FUNCTION F_Counter : BOOL

VAR_INPUT
	eCounterMode : E_CounterMode;
END_VAR
VAR_IN_OUT
	stCounter	: ST_Counter_Item;//ST_Conunter;
END_VAR
VAR
END_VAR

IF (eCounterMode = E_CounterMode.eCounterMode_Ok_Up) THEN
	stCounter.nValueOk:=stCounter.nValueOk+1;
	stCounter.nValueSerialError:=0;
ELSIF (eCounterMode = E_CounterMode.eCounterMode_Ok_Down) THEN	
	stCounter.nValueOk:=stCounter.nValueOk-1;
ELSIF (eCounterMode = E_CounterMode.eCounterMode_Ok_Clear) THEN	
	stCounter.nValueOk:=0;		
ELSIF (eCounterMode = E_CounterMode.eCounterMode_Nok_Up) THEN	
	stCounter.nValueNok:=stCounter.nValueNok+1;	
	stCounter.nValueSerialError:=stCounter.nValueSerialError+1;
ELSIF (eCounterMode = E_CounterMode.eCounterMode_Nok_Down) THEN	
	stCounter.nValueNok:=stCounter.nValueNok-1;	
ELSIF (eCounterMode = E_CounterMode.eCounterMode_Nok_Clear) THEN	
	stCounter.nValueNok:=0;	
ELSIF (eCounterMode = E_CounterMode.eCounterMode_SerialError_Clear) THEN	
	stCounter.nValueSerialError:=0;		
ELSIF (eCounterMode = E_CounterMode.eCounterMode_All_Clear) THEN	
	stCounter.nValueOk:=0;
	stCounter.nValueNok:=0;
	stCounter.nValueSerialError:=0;			
END_IF

END_FUNCTION

(* stored: Version 1.1.0.1, ProductVersion 3.1.4024.12
   POU F_Counter: Id {3642dcbf-67d5-401d-b611-819404e4eadf}, SpecialFunc None *)
